# EPICS substitutions: evrSupport/Db/ioc/IOC-IN20-MC01pattern.substitutions
#
# Pattern records
file evrPatternAll.db {
#	    Device        ,  SLC Pattern Check LNK    , EVR/Trigger
#	                                                  Links
  pattern { DEVICE        ,        LINK4              , LINK5 , LINK6 , TREF }
	  { IOC:IN20:MC01 ,         ""                ,  ""   ,  ""   , 1.03E06 }
}
file evrEventAll.db {
  pattern { DEVICE        }
	  { IOC:IN20:MC01 }
}
